{attribute 'linkalways'} 
{attribute 'no_explicit_call' := 'This FB is a CLASS and must be accessed using methods or properties'}
{attribute 'enable_dynamic_creation'}
FUNCTION_BLOCK _ETcVnSignedNormalization EXTENDS EnumDatatypeBase
VAR
	localData : ETcVnSignedNormalization;
	activeData : REFERENCE TO ETcVnSignedNormalization;
	enumBaseDatatype : _INT(localData);
END_VAR

METHOD PRIVATE AddLocalEnumeration
VAR_INPUT
	Enumeration : T_MAXSTRING;
	Value : ETcVnSignedNormalization;
END_VAR
AddEnumeration(Enumeration, Value);
END_METHOD

PROPERTY PUBLIC Address : PVOID
GET
Address := ADR(activeData);
END_GET
END_PROPERTY

METHOD PUBLIC ClearReference
VAR_INPUT
END_VAR
activeData REF= localData;
SetBaseDatatypeReference();
END_METHOD

METHOD PUBLIC Clone : I_Datatype
VAR
    pClone : POINTER TO _ETcVnSignedNormalization;
END_VAR
pClone := __NEW(_ETcVnSignedNormalization(InitialValue := Value));
Clone := pClone^;
END_METHOD

METHOD FB_init : BOOL
VAR_INPUT
	bInitRetains : BOOL; // if TRUE, the retain variables are initialized (warm start / cold start)
	bInCopyCode : BOOL;  // if TRUE, the instance afterwards gets moved into the copy code (online change)
	InitialValue : ETcVnSignedNormalization;
END_VAR
localData := InitialValue;
AddBaseDatatype(enumBaseDatatype);
ClearReference();

AddLocalEnumeration('TCVN_SN_FIX_ZERO', ETcVnSignedNormalization.TCVN_SN_FIX_ZERO);
AddLocalEnumeration('TCVN_SN_FULL_SCALE', ETcVnSignedNormalization.TCVN_SN_FULL_SCALE);
END_METHOD

PROPERTY PUBLIC Identifier : T_MAXSTRING
GET
Identifier := 'ETcVnSignedNormalization';
END_GET
END_PROPERTY

METHOD IsEnumeratorValueEqual : BOOL
VAR_INPUT
	Enumerator : I_KeyValueForwardEnumerator;
END_VAR
VAR
	storedValue : ETcVnSignedNormalization;
END_VAR
IF NOT Enumerator.TryGet(storedValue) THEN
	RETURN;
END_IF

IsEnumeratorValueEqual := storedValue = activeData;
END_METHOD

METHOD PUBLIC MakeReferenceTo
VAR_INPUT
	ReferenceTarget : REFERENCE TO ETcVnSignedNormalization;
END_VAR
activeData REF= ReferenceTarget;
SetBaseDatatypeReference();
END_METHOD

METHOD PROTECTED SetBaseDatatypeReference
VAR_INPUT
END_VAR
enumBaseDatatype.MakeReferenceTo(activeData);
END_METHOD

PROPERTY PUBLIC Size : UDINT
GET
Size := SIZEOF(activeData);
END_GET
END_PROPERTY

METHOD TryMakeReferenceTo : BOOL
VAR_INPUT
	Target : I_Datatype;
END_VAR
VAR
	targetAsEnum : I_EnumDatatype;
	pTargetData : POINTER TO ETcVnSignedNormalization;
END_VAR
IF NOT Target.TryResolveAsEnumDatatype(targetAsEnum) THEN
	RETURN;
END_IF

IF targetAsEnum.Identifier <> Identifier THEN
	RETURN;
END_IF

pTargetData := Target.Address;
activeData REF= pTargetData^;
SetBaseDatatypeReference();
TryMakeReferenceTo := TRUE;
END_METHOD

PROPERTY PUBLIC Value : ETcVnSignedNormalization
GET
Value := activeData;
END_GET
SET
activeData := Value;
END_SET
END_PROPERTY

END_FUNCTION_BLOCK

(* stored: Version 1.1.0.1, ProductVersion 3.1.4024.12
   POU _ETcVnSignedNormalization: Id {568decf6-b2c8-4448-9c4d-d1be69989e6f}, SpecialFunc None
   Folder Constructor: Id {a2e8718b-ef90-4277-a21a-6520c271359a}
   Folder Private: Id {4e4b162d-8a7b-4f98-bced-ffd4cc30e847}
   Folder Protected: Id {285174f6-99fe-408d-873f-be63f4c7ee40}
   Method AddLocalEnumeration: Id {9ffb9b92-49b0-4198-b1d7-c5253fccc379}
   Property Address: Id {9f4f9877-72bb-4bb8-a4cd-d87226a36989}
   Get Get: Id {9a3e87fe-beef-444e-bb79-31f36c430970}
   Method ClearReference: Id {25bb6d72-2cfd-494b-b862-6f0b68c6cada}
   Method Clone: Id {dd6313b4-aa71-456a-bcdf-f68f37f67409}
   Method FB_init: Id {988203c2-bfe6-4fae-82bc-9794347ddc31}
   Property Identifier: Id {b2f6f9fa-21ba-4c7f-82e1-926950e397c7}
   Get Get: Id {fe8ea72a-873d-455a-a1fa-b4cf44f9ec86}
   Method IsEnumeratorValueEqual: Id {0e151813-7202-4867-bb23-4801eac2f144}
   Method MakeReferenceTo: Id {9e87321a-a378-4f20-9a77-6b5c9f8ff497}
   Method SetBaseDatatypeReference: Id {3b67a01d-1453-455b-908b-f1a01f8d1bfb}
   Property Size: Id {fa68c4b8-cf9e-4e68-8e3c-9e54dd72806e}
   Get Get: Id {2f6a0595-ded1-4c2a-ae12-7042a56f3c15}
   Method TryMakeReferenceTo: Id {7d405a02-f28d-46df-8295-80e76d07af60}
   Property Value: Id {550b698d-764a-493b-a59b-c2561628cf4e}
   Get Get: Id {b3cb85ef-5ee5-4ec4-b884-815f5363244b}
   Set Set: Id {4d34a061-85dd-4d4f-900b-248d86b392e9} *)
